            mdesc nom_speed = {accel=200, vel=450, decel=200, tmax=2000, leave=30, reach=30}
            bool toStop
      [6]
        num nType
        pointRx pCircle = {fatherId=tTraj["test"].fFrame[0]}
        pointRx pPoint = {x=1198, y=151.559856, z=210.59, rx=87.981257, ry=172.229649, rz=-80.060298, fatherId=tTraj["test"].fFrame[0]}
        TrajectoryItem tSuper
          [0]
            string comment
            num distance
            InstrItem iInstr[3]
              [0]
                string sData
                string sType
              [1]
                string sData
                string sType
              [2]
                string sData
                string sType
            num moveType = 1
            num nMoveId
            num nStop
            num nTcpAction
            num nTime
            mdesc nom_speed = {accel=200, vel=450, decel=200, tmax=2000, blend=off}
            bool toStop = true

--- link_it.pgx ---
public program link_it(string x_sName)
begin
  // link all the point
  call link_all(x_sName)
  // put the base config
  tTraj[x_sName].tData[0].tSuper.moveType=1
end
